{attribute 'qualified_only'}
{attribute 'strict'}
TYPE ProcessSeq :
(
	NA := 0,
	Level10Done := 10,
	Level20Done := 20,
	Level30Done := 30,
	Level35Done := 35,	
	Level40Done := 40
);
END_TYPE

(* stored: Version 1.1.0.1, ProductVersion 3.1.4022.17
   EnumerationTextList ProcessSeq: Id {9040e6c5-0511-4467-a003-944a89ff5a0c} *)
